(*
SPDX-FileCopyrightText: © 2026 Oleksandr Tiutyk <trofimich@gmail.com>
SPDX-License-Identifier: MIT
License: https://opensource.org/license/mit
*)

{attribute 'qualified_only'}
{attribute 'strict'}
{attribute 'to_string'}
TYPE COMPARISION_RESULT :
(
	FIRST_LESS_THAN_SECOND := -1,
	FIRST_EQUAL_TO_SECOND := 0,
	FIRST_GREATER_THAN_SECOND := 1
) SINT;
END_TYPE

(* stored: Version 1.1.0.1
   DUT COMPARISION_RESULT: Id {15163b0f-b190-4edc-baf0-5adafd875cef} *)
